PROGRAM P5_01_EnableControls
VAR
	tonDisableNext			:TON;
	tonDisablePrev			:TON;
END_VAR
VAR // added by the converter: edge detectors and wires of the graphical bodies
    _w1, _w2 : BOOL;
END_VAR

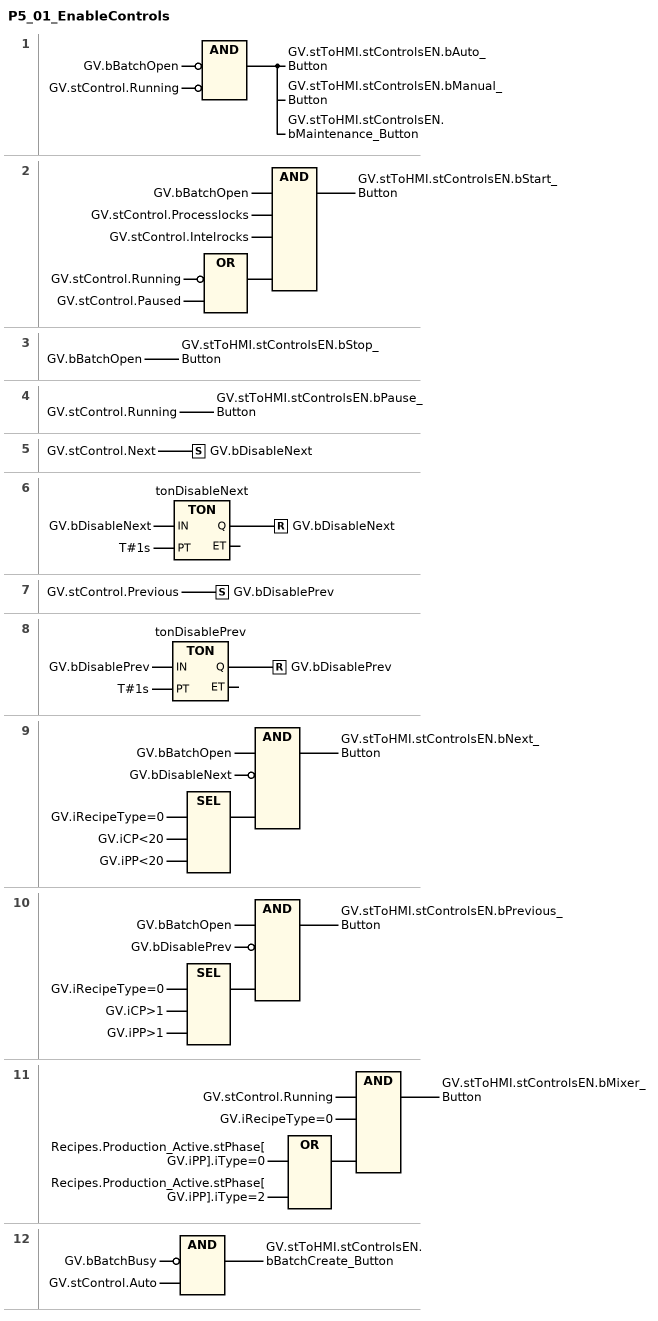
// NETWORK 1
_w1 := NOT GV.bBatchOpen AND NOT GV.stControl.Running;
GV.stToHMI.stControlsEN.bAuto_Button := _w1;
GV.stToHMI.stControlsEN.bManual_Button := _w1;
GV.stToHMI.stControlsEN.bMaintenance_Button := _w1;

// NETWORK 2
GV.stToHMI.stControlsEN.bStart_Button := GV.bBatchOpen AND GV.stControl.Processlocks AND GV.stControl.Intelrocks AND (NOT GV.stControl.Running OR GV.stControl.Paused);

// NETWORK 3
GV.stToHMI.stControlsEN.bStop_Button := GV.bBatchOpen;

// NETWORK 4
GV.stToHMI.stControlsEN.bPause_Button := GV.stControl.Running;

// NETWORK 5
GV.bDisableNext S= GV.stControl.Next;

// NETWORK 6
tonDisableNext(IN := GV.bDisableNext, PT := T#1s); // TON
GV.bDisableNext R= tonDisableNext.Q;

// NETWORK 7
GV.bDisablePrev S= GV.stControl.Previous;

// NETWORK 8
tonDisablePrev(IN := GV.bDisablePrev, PT := T#1s); // TON
GV.bDisablePrev R= tonDisablePrev.Q;

// NETWORK 9
GV.stToHMI.stControlsEN.bNext_Button := GV.bBatchOpen AND NOT GV.bDisableNext AND SEL(GV.iRecipeType=0, GV.iCP<20, GV.iPP<20);

// NETWORK 10
GV.stToHMI.stControlsEN.bPrevious_Button := GV.bBatchOpen AND NOT GV.bDisablePrev AND SEL(GV.iRecipeType=0, GV.iCP>1, GV.iPP>1);

// NETWORK 11
GV.stToHMI.stControlsEN.bMixer_Button := GV.stControl.Running AND (GV.iRecipeType=0) AND ((Recipes.Production_Active.stPhase[GV.iPP].iType=0) OR (Recipes.Production_Active.stPhase[GV.iPP].iType=2));

// NETWORK 12
GV.stToHMI.stControlsEN.bBatchCreate_Button := NOT GV.bBatchBusy AND GV.stControl.Auto;

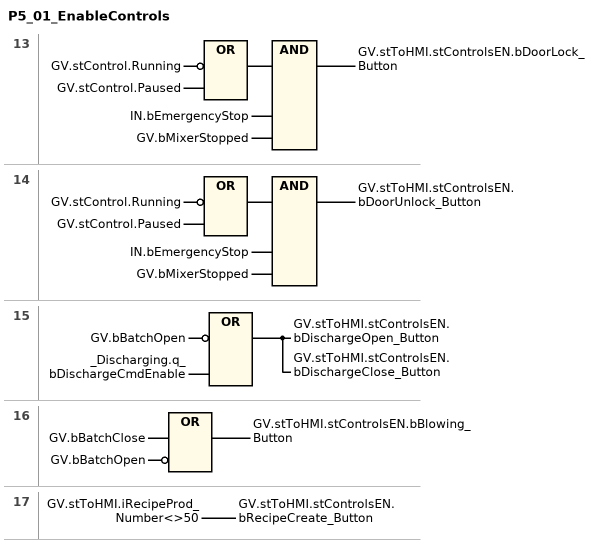
// NETWORK 13
GV.stToHMI.stControlsEN.bDoorLock_Button := (NOT GV.stControl.Running OR GV.stControl.Paused) AND IN.bEmergencyStop AND GV.bMixerStopped;

// NETWORK 14
GV.stToHMI.stControlsEN.bDoorUnlock_Button := (NOT GV.stControl.Running OR GV.stControl.Paused) AND IN.bEmergencyStop AND GV.bMixerStopped;

// NETWORK 15
_w2 := NOT GV.bBatchOpen OR _Discharging.q_bDischargeCmdEnable;
GV.stToHMI.stControlsEN.bDischargeOpen_Button := _w2;
GV.stToHMI.stControlsEN.bDischargeClose_Button := _w2;

// NETWORK 16
GV.stToHMI.stControlsEN.bBlowing_Button := GV.bBatchClose OR NOT GV.bBatchOpen;

// NETWORK 17
GV.stToHMI.stControlsEN.bRecipeCreate_Button := GV.stToHMI.iRecipeProd_Number<>50;

END_PROGRAM

(* stored: Version 1.1.0.1
   POU P5_01_EnableControls: Id {03708f81-cf31-4f21-abf9-33628c5a6011}, SpecialFunc None *)
